PROGRAM MAIN
VAR
	nSample				: UDINT;
	
	fbSource			: FB_CMA_Source := (	stInitPars 	:= cInitSource, 
												nOwnID 		:= eID_Source, 
												aDestIDs 	:= [eID_MagSpectrum,
																eID_EnvSpectrum,
																eID_Env,
																eID_RMS]);		
										
	fbSinkMagSpec		: FB_CMA_Sink 	:= ( 	nOwnID 		:= eID_MagSpec_Sink);
	fbSinkEnvSpec		: FB_CMA_Sink 	:= ( 	nOwnID 		:= eID_EnvSpec_Sink);
	fbSinkEnv			: FB_CMA_Sink 	:= ( 	nOwnID 		:= eID_Env_Sink);
	fbSinkRMS			: FB_CMA_Sink 	:= ( 	nOwnID 		:= eID_RMS_Sink); 
	
	nChannelIdx			: UDINT;

	k, m, l: UDINT;
	nChnIdx: UDINT;
END_VAR

Source();
Sink();
// input from EL3632
FOR nChannelIdx := 1 TO cMaxChannels DO
	FOR k := 1 TO cOversamples DO
		aAccBuffer[nChannelIdx][k] 		:= INT_TO_LREAL(aEl3632[nChannelIdx][k])*(5/EXPT(2,15))/(0.1)*9.81;
	END_FOR	
END_FOR

ACTION Sink:
// Push results to sink

fbSinkMagSpec.Output2DStd(	pDataOut 	:= ADR(aMagSpecResult), 
					nDataOutSize 		:= SIZEOF(aMagSpecResult), 
					eElementType 		:= eMA_TypeCode_LREAL, 
					nOptionPars			:= 0);
				
fbSinkEnvSpec.Output2DStd(	pDataOut 	:= ADR(aEnvSpecResult), 
					nDataOutSize 		:= SIZEOF(aEnvSpecResult), 
					eElementType 		:= eMA_TypeCode_LREAL, 
					nOptionPars			:= 0); 
					
fbSinkEnv.Output2DStd(	pDataOut 		:= ADR(aEnvResult), 
					nDataOutSize 		:= SIZEOF(aEnvResult), 
					eElementType 		:= eMA_TypeCode_LREAL, 
					nOptionPars			:= 0); 								
				
fbSinkRMS.Output2DStd(	pDataOut 		:= ADR(aRMSResult), 
					nDataOutSize 		:= SIZEOF(aRMSResult), 
					eElementType 		:= eMA_TypeCode_LREAL, 
					nOptionPars			:= 0);
END_ACTION

ACTION Source:
fbSource.Input2DStd( pDataIn 			:= ADR(aAccBuffer),
				  nDataInSize 			:= SIZEOF(aAccBuffer), 
				  eElementType 			:= eMA_TypeCode_LREAL,
				  nOptionPars			:= cCMA_Option_MarkInterruption );
END_ACTION

END_PROGRAM

(* stored: Version 1.1.0.1, ProductVersion 3.1.4024.12
   POU MAIN: Id {f43e4d9a-cbdc-4819-b719-b866da5ea61a}, SpecialFunc None
   Action Sink: Id {8275253b-e5d2-4fce-8863-ef6bc3f3c7a7}
   Action Source: Id {61bbab0f-1f8f-4023-aa28-0a5332181413} *)
